// TIA Portal V20 export
TYPE "typeReadVGageProData"
   STRUCT
      heartbeatActive : Bool;
      dataCollected : Bool;
      plcOK : Bool;
      spareIn_1 : Bool;
      spareIn_2 : Bool;
      spareIn_3 : Bool;
      spareIn_4 : Bool;
      spareIn_5 : Bool;
   END_STRUCT;
END_TYPE
